(* IEC 61131-3 sources: collections/test/List, 3 files *)

(* ---- Example.st ---- *)
USING AxUnit.Assert;

NAMESPACE Simatic.Ax.Collections

    // Example of a concrete customized ListItem
    CLASS MinMaxItem
        EXTENDS ListItem
        VAR PUBLIC
            Min : INT;
            Max : INT;
        END_VAR
    END_CLASS

    // Example of a concrete customized ListItem
    CLASS RangeItem
        EXTENDS ListItem
        VAR PUBLIC
            FromValue : INT;
            ToValue : INT;
        END_VAR
    END_CLASS

    {TestFixture}
    CLASS Example
        VAR PRIVATE
            _list : LinkedList;
            _i1 : MinMaxItem := (Min := 1, Max := 100);
            _i2 : MinMaxItem := (Min := 2, Max := 200);
            _i3 : RangeItem := (FromValue := 3, ToValue := 300); // declare a wrong, another list item which is not of type MinMaxItem
            _item : REF_TO MinMaxItem;
        END_VAR
        // Add 2 elements of MinMaxItem and one wrong element RangeItem to the list.
        // By reading the tail, the assignment attempt (?=) fails, because RangeItem can not be converted to MinMaxItem

        {Test}
        METHOD PUBLIC Test_Add_3_Elements_To_Queue_And_Get_Values_from_first_item
            _list.Add(item := _i1); // add i1 to head
            _list.Add(item := _i2);
            _list.Add(item := _i3); // add _i3, a wrong IListItem to the list (Tail)
            _item ?= _list.Tail(); // assignment attempt (?=) --> It's NULL if not of type MinMaxItem
            Equal(_item <> NULL, TRUE);
            IF (_item <> NULL) THEN
                Equal(_item^.Min, 1);
                Equal(_item^.Max, 100);
            END_IF;
            _item ?= _list.Head(); // assignment attempt (?=) --> It's NULL if not of type MinMaxItem
            Equal(_item = NULL, TRUE);
            IF (_item <> NULL) THEN
                NotEqual(_item^.Min, 3);
                NotEqual(_item^.Max, 300);
            END_IF;
            Equal(expected := 3, actual := _list.Count());
        END_METHOD
    END_CLASS

END_NAMESPACE

(* ---- TestList.st ---- *)
USING AxUnit.Assert;
USING Simatic.Ax.Collections;
USING AxUnit.Assert;

NAMESPACE Simatic.Ax.Collections
    {TestFixture}
    CLASS TestList
        VAR PRIVATE
            _list : LinkedList;
            _i1 : ListItem;
            _i2 : ListItem;
            _i3 : ListItem;
            _ifake : ListItem;
            _iReturn : IListItem;
            _item : IListItem;
        END_VAR

        {Test}
        METHOD PUBLIC Test_Add_Expect_Item
            _item := _i1;
            _iReturn := _list.Add(item := _i1);
            Equal(_iReturn = _item, TRUE);
            Equal(_list.Count(), 1);
        END_METHOD

        {Test}
        METHOD PUBLIC Test_Add_3_Elements
            _iReturn := _list.Add(item := _i1);
            _iReturn := _list.Add(item := _i2);
            _iReturn := _list.Add(item := _i3);

            _item := _i3; // Tail
            Equal(_list.Head() = _item, TRUE);

            _item := _i1; // Tail
            Equal(_list.Tail() = _item, TRUE);

            Equal(_list.Count(), 3);
        END_METHOD

        {Test}
        METHOD PUBLIC Test_Tail_Top_NULL
            THIS.Test_Add_3_Elements();
            Equal(_list.Tail().PreviousItem() = NULL, TRUE);
            Equal(_list.Head().NextItem() = NULL, TRUE);
        END_METHOD
        {Test}

        METHOD PUBLIC Test_Tail_Next_Equals_Top
            _list.Add(item := _i1);
            _list.Add(item := _i2);
            _list.Add(item := _i3, join := TRUE);

            _item := _i1;
            Equal(_list.Head().NextItem() = _item, TRUE);

            _item := _i3;
            Equal(_list.Tail().PreviousItem() = _item, TRUE);
        END_METHOD

        {Test}
        METHOD PUBLIC Test_RemoveItem_i2_and_expect_i1_i3_linked
            THIS.Test_Add_3_Elements();

            _list.Remove(_i2);
            _item := _i1;
            Equal(_list.Head().PreviousItem() = _item, TRUE);
            _item := _i3;
            Equal(_list.Tail().NextItem() = _item, TRUE);
        END_METHOD

        {Test}
        METHOD PUBLIC Test_RemoveItem_tail_and_expect_i2_tail
            VAR_TEMP
                result : BOOL;
            END_VAR
            THIS.Test_Add_3_Elements();

            result := _list.Remove(_list.Tail());
            _item := _i2;
            Equal(result, TRUE);
            Equal(_list.Tail() = _item, TRUE);
            Equal(_list.Tail().PreviousItem() = NULL, TRUE);
        END_METHOD

        {Test}
        METHOD PUBLIC Test_RemoveItem_head_and_expect_i2_head
            VAR_TEMP
                result : BOOL;
            END_VAR

            THIS.Test_Add_3_Elements();

            result := _list.Remove(_list.Head());
            _item := _i2;
            Equal(result, TRUE);
            Equal(_list.Head() = _item, TRUE);
            Equal(_list.Head().NextItem() = NULL, TRUE);
        END_METHOD

        {Test}
        METHOD PUBLIC Test_RemoveAllItems_and_Expect_tail_and_head_null
            VAR_TEMP
                result : BOOL;
            END_VAR
            THIS.Test_Add_3_Elements();

            _list.Remove(_list.Head());
            _list.Remove(_list.Head());
            result := _list.Remove(_list.Head());

            Equal(result, TRUE);
            Equal(_list.Head() = NULL, TRUE);
            Equal(_list.Tail() = NULL, TRUE);
        END_METHOD

        {Test}
        METHOD PUBLIC Remove_From_Empty_List_and_expect_false
            Equal(_list.Remove(_i1), FALSE);
        END_METHOD

        {Test}
        METHOD PUBLIC Remove_NotExisting_item_from_list_and_expect_false
            THIS.Test_Add_3_Elements();
            Equal(_list.Remove(_ifake), FALSE);
        END_METHOD
    END_CLASS
END_NAMESPACE

(* ---- TestStack.st ---- *)
USING AxUnit.Assert;
USING Simatic.Ax.Collections;
USING AxUnit.Assert;

NAMESPACE Simatic.Ax.Collections
    {TestFixture}
    CLASS TestStack
        VAR PRIVATE
            _stack : Stack;
            _stackStateLess : Stack;
            _i1 : ListItem;
            _i2 : ListItem;
            _i3 : ListItem;
            _ifake : ListItem;
            _iReturn : IListItem;
            _item : IListItem;
        END_VAR

        // This method will be called before each test method
        {TestSetup}
        METHOD PUBLIC MyTestSetup
            _stack := _stackStateLess;
        END_METHOD

        {Test}
        METHOD PUBLIC Test_Add_Expect_Item
            _item := _i1;
            _iReturn := _stack.Push(item := _i1);
            Equal(_iReturn = _item, TRUE);
            Equal(_stack.Count(), 1);
        END_METHOD

        {Test}
        METHOD PUBLIC Test_Add_3_Elements
            _iReturn := _stack.Push(item := _i1);
            _iReturn := _stack.Push(item := _i2);
            _iReturn := _stack.Push(item := _i3);

            _item := _i3;
            Equal(_stack.Peek() = _item, TRUE);
            Equal(_stack.Count(), 3);
        END_METHOD

        {Test}
        METHOD PUBLIC Test_Top_NULL
            THIS.Test_Add_3_Elements();
            Equal(_stack.Peek().NextItem() = NULL, TRUE);
        END_METHOD

        {Test}
        METHOD PUBLIC Test_PopItem_and_expect_i3_and_i2_on_top
            THIS.Test_Add_3_Elements();

            _item := _i3;
            Equal(_stack.Pop() = _item, TRUE);
            _item := _i2;
            Equal(_stack.Peek() = _item, TRUE);
        END_METHOD

        {Test}
        METHOD PUBLIC Test_Pop_2_Items_and_expect_i2_and_i1_on_top

            THIS.Test_Add_3_Elements();

            _item := _i2;
            _stack.Pop();
            Equal(_stack.Pop() = _item, TRUE);

            _item := _i1;
            Equal(_stack.Peek() = _item, TRUE);
        END_METHOD

        {Test}
        METHOD PUBLIC Test_Pop_from_empty_List
            Equal(_stack.Pop() = NULL, TRUE);
        END_METHOD

    END_CLASS
END_NAMESPACE
